PROGRAM LoadModel
VAR
	bDone : BOOL;
	iPrediction : INT;
END_VAR

VAR_INPUT
	bPython : BOOL;
END_VAR

IF bPython THEN
	IF bDone THEN
		bPython := FALSE;
		bDone := FALSE;
	END_IF
END_IF

END_PROGRAM

(* stored: Version 1.1.0.1, ProductVersion 3.1.4024.9
   POU LoadModel: Id {2c3102db-f6b6-4a4e-b1bf-97c6dc05c8fb}, SpecialFunc None *)
